{attribute 'qualified_only'}
VAR_GLOBAL
	// Main funktioner //
	bPowerOn			:	BOOL;
	bPowerOff			:	BOOL;
	bEmergency			:	BOOL;
	bAutomaticMode		:	BOOL;
	bKapsekvens			:	BOOL;
	bKapsekvensDone		:	BOOL;

	// Svärd hållare //
	bSvard1				:	BOOL;
	bSvard2				:	BOOL;
	bSvardVentil1		:	BOOL;
	bSvardVentil2		:	BOOL;
	bSvard1Last			:	BOOL;
	bSvard1EjLast		:	BOOL;
	bSvard2Last			:	BOOL;
	bSvard2EjLast		:	BOOL;
	
	// Renhållning av maskin //
	bRenblasningsVentil	:	BOOL;
	Span_trans_Timer	: TOF;
	
	// Motor kontroller //
	bSagblad			:	BOOL;
	bKylpump			:	BOOL;
	
END_VAR

(* stored: Version 1.1.0.1, ProductVersion 3.1.4024.10
   GVL GVL: Id {23e81069-fc6f-4f01-b242-7f728f6bb6bc} *)
